# EPICS autosave request: ADApp/Db/prosilica_settings.req
$(P)$(R)PSReadStatistics.SCAN
$(P)$(R)PSByteRate
$(P)$(R)PSPacketSize
$(P)$(R)SyncOut1Mode
$(P)$(R)SyncOut1Level
$(P)$(R)SyncOut1Invert
$(P)$(R)SyncOut2Mode
$(P)$(R)SyncOut2Level
$(P)$(R)SyncOut2Invert
$(P)$(R)SyncOut3Mode
$(P)$(R)SyncOut3Level
$(P)$(R)SyncOut3Invert
$(P)$(R)Strobe1Mode
$(P)$(R)Strobe1CtlDuration
$(P)$(R)Strobe1Delay
$(P)$(R)Strobe1Duration
$(P)$(R)TriggerEvent
$(P)$(R)TriggerOverlap
$(P)$(R)TriggerDelay
